Staubli VAL3: loadFile.pgx

public program loadFile(num x_nCamID (dimensions=1), string x_sNameJob (dimensions=1), bool& x_bError[] (dimensions=1))
begin
  //-----------------------------------------------------------------------
  //Header begin
  //Description of program
  //  Loads the specified job from flash memory on the In-Sight sensor,
  //  making it the active job.
  //
  //!!! The In-Sight sensor must be OFFLINE !!!
  //
  //Input parameters
  //  num x_nCamID :
  //    role : camera's ID
  //
  //Output parameters
  //  string x_sNameJob :
  //    role : The name of the job.
  //           The command will execute with or without the .JOB extension.
  //
  //  bool x_bError :
  //    role : returns true if an error occurred and false otherwise
  //
  //Examples
  //   call loadFile(nCamID,"Camera1.job",x_bError)
  //
  //History
  //  Creation : 19-05-08 - f.Rob
  //Header end
  //-----------------------------------------------------------------------

  nProgram[x_nCamID]=4
  call sendCommand(x_nCamID,"LF"+x_sNameJob,x_bError)
end
